SYSTEM System
  DEVICE DEV0 : NXT_RMTDEV(WATCH_ID := localhost:61497, HMI_ID := localhost:61498, MGR_ID := localhost:61499)
    RESOURCE RES0 : EMB_RES
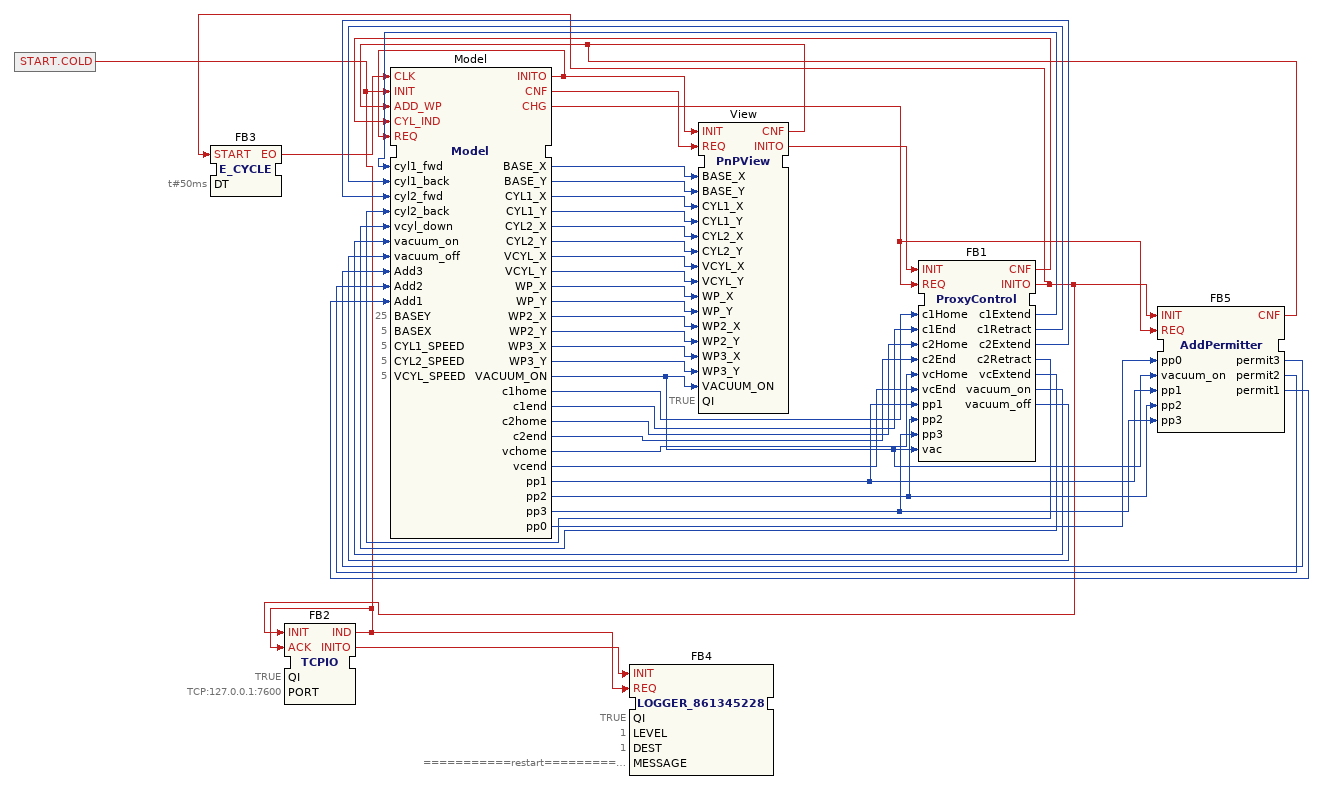
      FBS
        FB3 : E_CYCLE(DT := t#50ms);
        View : PnPView(QI := TRUE);
        FB1 : ProxyControl;
        FB2 : TCPIO(QI := TRUE, PORT := TCP:127.0.0.1:7600);
        FB4 : LOGGER_861345228(QI := TRUE, LEVEL := 1, DEST := 1, MESSAGE := ===========restart===========); {SET_ATTRIBUTE(Configuration.GenericFBType.InterfaceParams, Runtime.System#CNT:=1)}
        Model : Model(BASEY := 25, BASEX := 5, CYL1_SPEED := 5, CYL2_SPEED := 5, VCYL_SPEED := 5);
        FB5 : AddPermitter;
      END_FBS
      EVENT_CONNECTIONS
        FB3.EO TO Model.CLK;
        START.COLD TO Model.INIT;
        Model.INITO TO View.INIT;
        Model.CNF TO View.REQ;
        View.CNF TO Model.ADD_WP;
        View.INITO TO FB1.INIT;
        Model.CHG TO FB1.REQ;
        FB1.CNF TO Model.CYL_IND;
        FB1.INITO TO FB3.START;
        FB1.INITO TO FB2.INIT;
        FB2.IND TO Model.INIT;
        FB2.IND TO FB2.ACK;
        FB2.INITO TO FB4.INIT;
        FB2.IND TO FB4.REQ;
        FB1.INITO TO FB5.INIT;
        FB5.CNF TO Model.ADD_WP;
        Model.CHG TO FB5.REQ;
        Model.INITO TO Model.REQ;
      END_CONNECTIONS
      DATA_CONNECTIONS
        Model.BASE_X TO View.BASE_X;
        Model.BASE_Y TO View.BASE_Y;
        Model.CYL1_X TO View.CYL1_X;
        Model.CYL1_Y TO View.CYL1_Y;
        Model.CYL2_X TO View.CYL2_X;
        Model.CYL2_Y TO View.CYL2_Y;
        Model.VCYL_X TO View.VCYL_X;
        Model.VCYL_Y TO View.VCYL_Y;
        Model.WP_X TO View.WP_X;
        Model.WP_Y TO View.WP_Y;
        Model.WP2_X TO View.WP2_X;
        Model.WP2_Y TO View.WP2_Y;
        Model.WP3_X TO View.WP3_X;
        Model.WP3_Y TO View.WP3_Y;
        Model.VACUUM_ON TO View.VACUUM_ON;
        Model.c1home TO FB1.c1Home;
        Model.c1end TO FB1.c1End;
        Model.c2home TO FB1.c2Home;
        Model.c2end TO FB1.c2End;
        Model.vchome TO FB1.vcHome;
        Model.vcend TO FB1.vcEnd;
        Model.pp1 TO FB1.pp1;
        Model.pp2 TO FB1.pp2;
        Model.pp3 TO FB1.pp3;
        Model.VACUUM_ON TO FB1.vac;
        FB1.c1Extend TO Model.cyl1_fwd;
        FB1.c1Retract TO Model.cyl1_back;
        FB1.c2Extend TO Model.cyl2_fwd;
        FB1.c2Retract TO Model.cyl2_back;
        FB1.vcExtend TO Model.vcyl_down;
        FB1.vacuum_on TO Model.vacuum_on;
        FB1.vacuum_off TO Model.vacuum_off;
        Model.pp0 TO FB5.pp0;
        Model.VACUUM_ON TO FB5.vacuum_on;
        Model.pp1 TO FB5.pp1;
        Model.pp2 TO FB5.pp2;
        Model.pp3 TO FB5.pp3;
        FB5.permit3 TO Model.Add3;
        FB5.permit2 TO Model.Add2;
        FB5.permit1 TO Model.Add1;
      END_CONNECTIONS
    END_RESOURCE
  END_DEVICE
END_SYSTEM
